// TIA Portal project "Pick And Place(Basic)" (V17)
// Vorlageprojekt für das Buch mit Zielsystem S7-1200

(* hardware
DEVICE "S7-1200-Station_1"  S7-1200 Station
   slot 0: "Baugruppenträger_0"  Rack  V1.0
   slot 1: "PLC_1"  CPU 1211C DC/DC/DC  6ES7 211-1AE40-0XB0  V4.1
*)

// ===== PLC "PLC_1"  CPU 1211C DC/DC/DC =====

VAR_GLOBAL   // PLC tag table "Standard-Variablentabelle"
   "system on" AT %M0.0 : Bool;
   "current steps" AT %MW3 : Int;
   "Tag_1" AT %M0.2 : Bool;
   "Tag_2" AT %M0.3 : Bool;
   "Tag_3" AT %M0.5 : Bool;
   "Tag_4" AT %M0.7 : Bool;
   "entry conveyor 2" AT %M7.0 : Bool;
   "entry conveyor 1" AT %M7.1 : Bool;
   "Tag_5" AT %M12.4 : Bool;
   "Tag_6" AT %M12.7 : Bool;
   "Tag_7" AT %M24.5 : Bool;
END_VAR

VAR_GLOBAL   // PLC tag table "Tag table from XML_1"
   "Item at entry" AT %I0.0 : Bool;
   "Item at exit" AT %I0.1 : Bool;
   "Moving X" AT %I0.2 : Bool;
   "Moving Z" AT %I0.3 : Bool;
   "Item detected" AT %I0.4 : Bool;
   "Start" AT %I0.5 : Bool;
   "Reset" AT %I0.6 : Bool;
   "Stop" AT %I0.7 : Bool;
   "Emergency stop" AT %I1.0 : Bool;
   "Auto" AT %I1.1 : Bool;
   "FACTORY I/O (Running)" AT %I1.2 : Bool;
   "Entry conveyor" AT %Q0.0 : Bool;
   "Exit conveyor" AT %Q0.1 : Bool;
   "Move X" AT %Q0.2 : Bool;
   "Move Z" AT %Q0.3 : Bool;
   "Grab" AT %Q0.4 : Bool;
   "Start light" AT %Q0.5 : Bool;
   "Reset light" AT %Q0.6 : Bool;
   "Stop light" AT %Q0.7 : Bool;
   "Counter" AT %QD30 : DInt;
END_VAR

FUNCTION "MHJ-PLC-Lab-Function-S71200" : Void   // FC9000, SCL
{ S7_Optimized_Access := 'TRUE' }
VERSION : 0.1
   VAR_TEMP
      rdTimeReturn : Int;
      outputTime : DTL;
      SyncVal : Byte;
      forVal : Int;
      forVal_2 : Int;
      Value : Byte;
   END_VAR
   VAR CONSTANT
      CompVal : Byte := 16#34;
      Value_01 : Byte := 16#11;
      Value_01_DW : DWord := 16#A165_D992;
      Value_02_DW : DWord := 16#58BE_4401;
   END_VAR
BEGIN

   #Value:=PEEK(area := 16#82,
        dbNumber := 0,
        byteOffset := 511);
   #Value := #Value + 1;

   POKE(area := 16#82,
        dbNumber := 0,
        byteOffset := 511,
        value := #Value);

   POKE(area:=16#81,
        dbNumber:=0,
        byteOffset:=1016,
        value:=#Value_01_DW);
   POKE(area := 16#81,
        dbNumber := 0,
        byteOffset := 1020,
        value := #Value_02_DW);

   POKE(area := 16#81,
        dbNumber := 0,
        byteOffset := 511,
        value := B#16#00);

   FOR #forVal := 0 TO 120 DO
       FOR #forVal_2:=0 TO 10 DO
           #rdTimeReturn:=RD_SYS_T(#outputTime);
           #rdTimeReturn := WR_SYS_T(#outputTime);
           #rdTimeReturn := RD_SYS_T(#outputTime);
           #rdTimeReturn := WR_SYS_T(#outputTime);
       END_FOR;
       #SyncVal:= PEEK(area := 16#81,
                      dbNumber := 0,
                      byteOffset := 511);
       IF #SyncVal = #CompVal THEN
          GOTO M_1;
       END_IF;
   END_FOR;
   RETURN;

   M_1:
   POKE(area := 16#81,
        dbNumber := 0,
        byteOffset := 511,
        value := B#16#0);
END_FUNCTION

ORGANIZATION_BLOCK "Main"   // OB1, LAD, ProgramCycle
TITLE = "Main Program Sweep (Cycle)"
{ S7_Optimized_Access := 'TRUE' }
VERSION : 0.1
   VAR_INPUT
      Initial_Call : Bool;   // Initial call of this OB
      Remanence : Bool;   // =True, if remanent data are available
   END_VAR
   VAR_TEMP   // added for the SCL form of the ladder/FBD networks
      _w1 : Bool;
      _w2 : Bool;
   END_VAR
BEGIN

REGION Network 1: Konnektierungsbaustein für PLC-Lab
   // Im Netzwerk 1 wird der Konnektierungsbaustein für PLC-Lab aufgerufen.
   // Dieser Aufruf darf nicht entfernt werden!
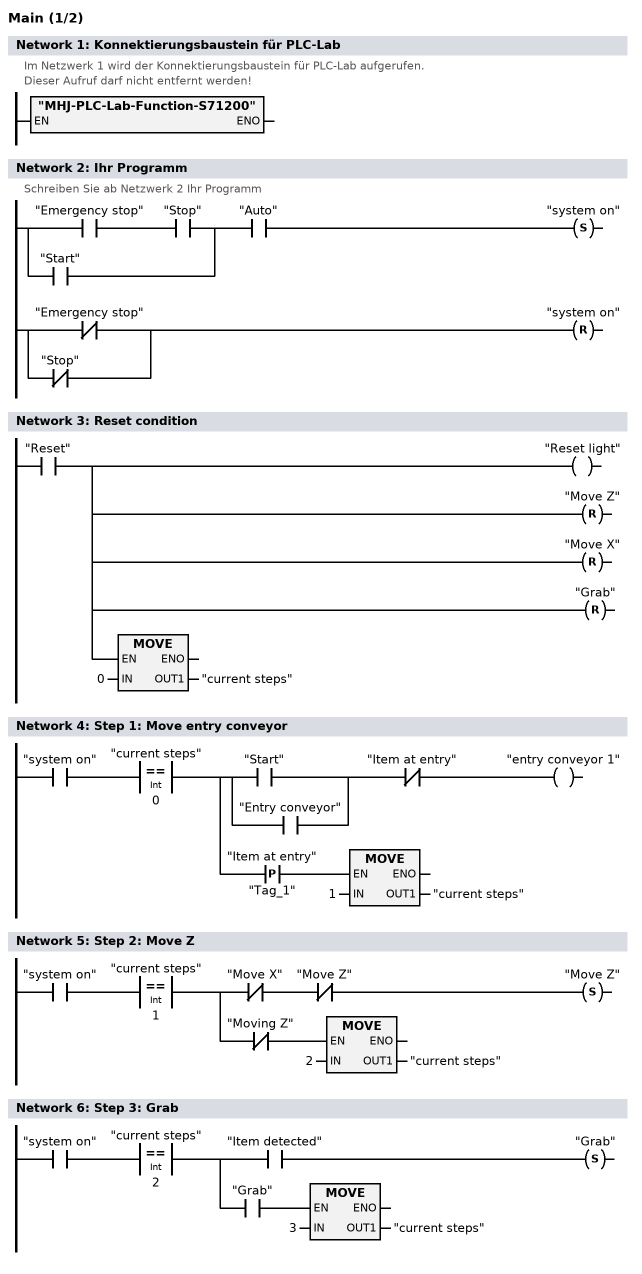
   RUNG wire#powerrail
      "MHJ-PLC-Lab-Function-S71200"()
   END_RUNG
   // the same network as SCL:
   "MHJ-PLC-Lab-Function-S71200"();
END_REGION

REGION Network 2: Ihr Programm
   // Schreiben Sie ab Netzwerk 2 Ihr Programm
   RUNG wire#powerrail
      Contact( "Emergency stop" )
      Contact( "Stop" )
      wire#w1
      Contact( "Auto" )
      S_Coil( "system on" )
   END_RUNG
   RUNG wire#powerrail
      Contact( "Start" )
   END_RUNG wire#w1
   RUNG wire#powerrail
      I_Contact( "Emergency stop" )
      wire#w2
      R_Coil( "system on" )
   END_RUNG
   RUNG wire#powerrail
      I_Contact( "Stop" )
   END_RUNG wire#w2
   // the same network as SCL:
   IF (("Emergency stop" AND "Stop") OR "Start") AND "Auto" THEN "system on" := TRUE; END_IF;
   IF NOT "Emergency stop" OR NOT "Stop" THEN "system on" := FALSE; END_IF;
END_REGION

REGION Network 3: Reset condition
   RUNG wire#powerrail
      Contact( "Reset" )
      wire#w1
      Coil( "Reset light" )
   END_RUNG
   RUNG wire#w1
      R_Coil( "Move Z" )
   END_RUNG
   RUNG wire#w1
      R_Coil( "Move X" )
   END_RUNG
   RUNG wire#w1
      R_Coil( "Grab" )
   END_RUNG
   RUNG wire#w1
      Move(in := 0, out1 => "current steps")
   END_RUNG
   // the same network as SCL:
   "Reset light" := "Reset";
   IF "Reset" THEN
       "Move Z" := FALSE;
       "Move X" := FALSE;
       "Grab" := FALSE;
       "current steps" := 0;
   END_IF;
END_REGION

REGION Network 4: Step 1: Move entry conveyor
   RUNG wire#powerrail
      Contact( "system on" )
      { S7_Templates := "SrcType := Int" } EQ_Contact(in1 := "current steps", in2 := 0)
      wire#w1
      Contact( "Start" )
      wire#w2
      I_Contact( "Item at entry" )
      Coil( "entry conveyor 1" )
   END_RUNG
   RUNG wire#w1
      Contact( "Entry conveyor" )
   END_RUNG wire#w2
   RUNG wire#w1
      P_Contact(operand := "Item at entry", bit := "Tag_1")
      Move(in := 1, out1 => "current steps")
   END_RUNG
   // the same network as SCL:
   #_w1 := "system on" AND ("current steps" = 0);
   "entry conveyor 1" := #_w1 AND ("Start" OR "Entry conveyor") AND NOT "Item at entry";
   #_w2 := #_w1 AND "Item at entry" AND NOT "Tag_1";   // rising edge of "Item at entry"
   "Tag_1" := "Item at entry";
   IF #_w2 THEN "current steps" := 1; END_IF;
END_REGION

REGION Network 5: Step 2: Move Z
   RUNG wire#powerrail
      Contact( "system on" )
      { S7_Templates := "SrcType := Int" } EQ_Contact(in1 := "current steps", in2 := 1)
      wire#w1
      I_Contact( "Move X" )
      I_Contact( "Move Z" )
      S_Coil( "Move Z" )
   END_RUNG
   RUNG wire#w1
      I_Contact( "Moving Z" )
      Move(in := 2, out1 => "current steps")
   END_RUNG
   // the same network as SCL:
   #_w1 := "system on" AND ("current steps" = 1);
   IF #_w1 AND NOT "Move X" AND NOT "Move Z" THEN "Move Z" := TRUE; END_IF;
   IF #_w1 AND NOT "Moving Z" THEN "current steps" := 2; END_IF;
END_REGION

REGION Network 6: Step 3: Grab
   RUNG wire#powerrail
      Contact( "system on" )
      { S7_Templates := "SrcType := Int" } EQ_Contact(in1 := "current steps", in2 := 2)
      wire#w1
      Contact( "Item detected" )
      S_Coil( "Grab" )
   END_RUNG
   RUNG wire#w1
      Contact( "Grab" )
      Move(in := 3, out1 => "current steps")
   END_RUNG
   // the same network as SCL:
   #_w1 := "system on" AND ("current steps" = 2);
   IF #_w1 AND "Item detected" THEN "Grab" := TRUE; END_IF;
   IF #_w1 AND "Grab" THEN "current steps" := 3; END_IF;
END_REGION

REGION Network 7: Step 4: Moving Z part 2
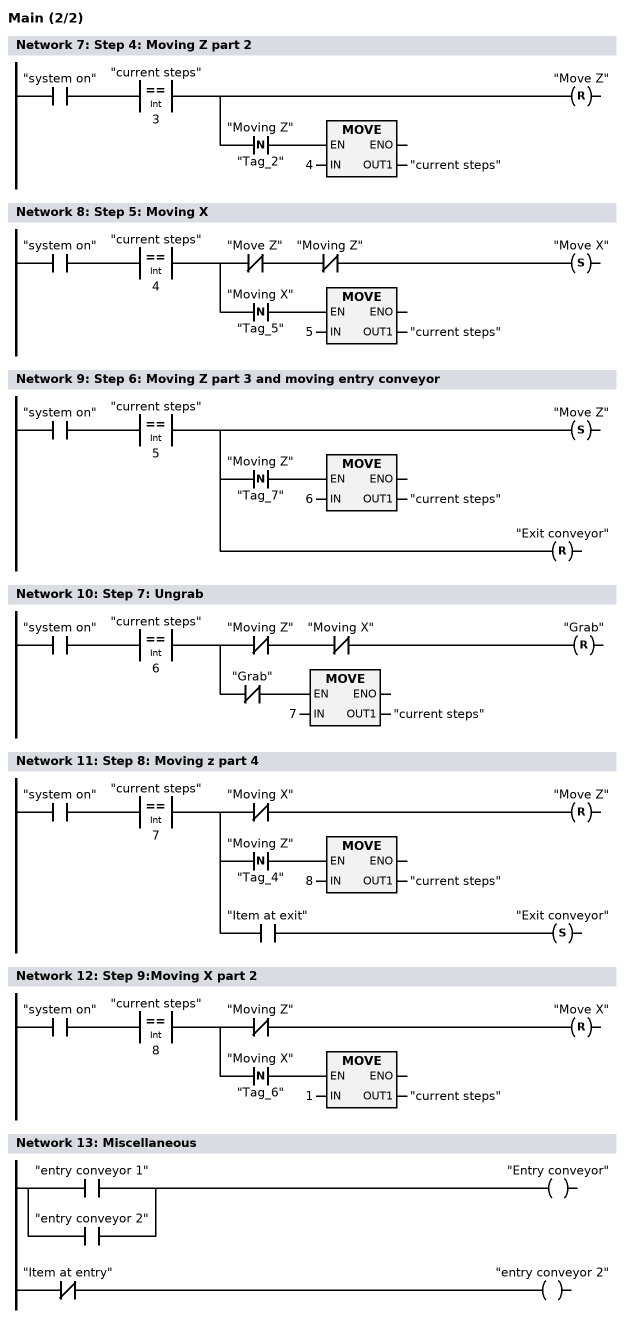
   RUNG wire#powerrail
      Contact( "system on" )
      { S7_Templates := "SrcType := Int" } EQ_Contact(in1 := "current steps", in2 := 3)
      wire#w1
      R_Coil( "Move Z" )
   END_RUNG
   RUNG wire#w1
      N_Contact(operand := "Moving Z", bit := "Tag_2")
      Move(in := 4, out1 => "current steps")
   END_RUNG
   // the same network as SCL:
   #_w1 := "system on" AND ("current steps" = 3);
   IF #_w1 THEN "Move Z" := FALSE; END_IF;
   #_w2 := #_w1 AND NOT "Moving Z" AND "Tag_2";   // falling edge of "Moving Z"
   "Tag_2" := "Moving Z";
   IF #_w2 THEN "current steps" := 4; END_IF;
END_REGION

REGION Network 8: Step 5: Moving X
   RUNG wire#powerrail
      Contact( "system on" )
      { S7_Templates := "SrcType := Int" } EQ_Contact(in1 := "current steps", in2 := 4)
      wire#w1
      I_Contact( "Move Z" )
      I_Contact( "Moving Z" )
      S_Coil( "Move X" )
   END_RUNG
   RUNG wire#w1
      N_Contact(operand := "Moving X", bit := "Tag_5")
      Move(in := 5, out1 => "current steps")
   END_RUNG
   // the same network as SCL:
   #_w1 := "system on" AND ("current steps" = 4);
   IF #_w1 AND NOT "Move Z" AND NOT "Moving Z" THEN "Move X" := TRUE; END_IF;
   #_w2 := #_w1 AND NOT "Moving X" AND "Tag_5";   // falling edge of "Moving X"
   "Tag_5" := "Moving X";
   IF #_w2 THEN "current steps" := 5; END_IF;
END_REGION

REGION Network 9: Step 6: Moving Z part 3 and moving entry conveyor
   RUNG wire#powerrail
      Contact( "system on" )
      { S7_Templates := "SrcType := Int" } EQ_Contact(in1 := "current steps", in2 := 5)
      wire#w1
      S_Coil( "Move Z" )
   END_RUNG
   RUNG wire#w1
      N_Contact(operand := "Moving Z", bit := "Tag_7")
      Move(in := 6, out1 => "current steps")
   END_RUNG
   RUNG wire#w1
      R_Coil( "Exit conveyor" )
   END_RUNG
   // the same network as SCL:
   #_w1 := "system on" AND ("current steps" = 5);
   IF #_w1 THEN "Move Z" := TRUE; END_IF;
   #_w2 := #_w1 AND NOT "Moving Z" AND "Tag_7";   // falling edge of "Moving Z"
   "Tag_7" := "Moving Z";
   IF #_w2 THEN "current steps" := 6; END_IF;
   IF #_w1 THEN "Exit conveyor" := FALSE; END_IF;
END_REGION

REGION Network 10: Step 7: Ungrab
   RUNG wire#powerrail
      Contact( "system on" )
      { S7_Templates := "SrcType := Int" } EQ_Contact(in1 := "current steps", in2 := 6)
      wire#w1
      I_Contact( "Moving Z" )
      I_Contact( "Moving X" )
      R_Coil( "Grab" )
   END_RUNG
   RUNG wire#w1
      I_Contact( "Grab" )
      Move(in := 7, out1 => "current steps")
   END_RUNG
   // the same network as SCL:
   #_w1 := "system on" AND ("current steps" = 6);
   IF #_w1 AND NOT "Moving Z" AND NOT "Moving X" THEN "Grab" := FALSE; END_IF;
   IF #_w1 AND NOT "Grab" THEN "current steps" := 7; END_IF;
END_REGION

REGION Network 11: Step 8: Moving z part 4
   RUNG wire#powerrail
      Contact( "system on" )
      { S7_Templates := "SrcType := Int" } EQ_Contact(in1 := "current steps", in2 := 7)
      wire#w1
      I_Contact( "Moving X" )
      R_Coil( "Move Z" )
   END_RUNG
   RUNG wire#w1
      N_Contact(operand := "Moving Z", bit := "Tag_4")
      Move(in := 8, out1 => "current steps")
   END_RUNG
   RUNG wire#w1
      Contact( "Item at exit" )
      S_Coil( "Exit conveyor" )
   END_RUNG
   // the same network as SCL:
   #_w1 := "system on" AND ("current steps" = 7);
   IF #_w1 AND NOT "Moving X" THEN "Move Z" := FALSE; END_IF;
   #_w2 := #_w1 AND NOT "Moving Z" AND "Tag_4";   // falling edge of "Moving Z"
   "Tag_4" := "Moving Z";
   IF #_w2 THEN "current steps" := 8; END_IF;
   IF #_w1 AND "Item at exit" THEN "Exit conveyor" := TRUE; END_IF;
END_REGION

REGION Network 12: Step 9:Moving X part 2
   RUNG wire#powerrail
      Contact( "system on" )
      { S7_Templates := "SrcType := Int" } EQ_Contact(in1 := "current steps", in2 := 8)
      wire#w1
      I_Contact( "Moving Z" )
      R_Coil( "Move X" )
   END_RUNG
   RUNG wire#w1
      N_Contact(operand := "Moving X", bit := "Tag_6")
      Move(in := 1, out1 => "current steps")
   END_RUNG
   // the same network as SCL:
   #_w1 := "system on" AND ("current steps" = 8);
   IF #_w1 AND NOT "Moving Z" THEN "Move X" := FALSE; END_IF;
   #_w2 := #_w1 AND NOT "Moving X" AND "Tag_6";   // falling edge of "Moving X"
   "Tag_6" := "Moving X";
   IF #_w2 THEN "current steps" := 1; END_IF;
END_REGION

REGION Network 13: Miscellaneous
   RUNG wire#powerrail
      Contact( "entry conveyor 1" )
      wire#w1
      Coil( "Entry conveyor" )
   END_RUNG
   RUNG wire#powerrail
      Contact( "entry conveyor 2" )
   END_RUNG wire#w1
   RUNG wire#powerrail
      I_Contact( "Item at entry" )
      Coil( "entry conveyor 2" )
   END_RUNG
   // the same network as SCL:
   "Entry conveyor" := "entry conveyor 1" OR "entry conveyor 2";
   "entry conveyor 2" := NOT "Item at entry";
END_REGION
END_ORGANIZATION_BLOCK